Omron Sysmac Studio project Major Project Group 6-week12_011125 (Sysmac Studio 1.56.0.64011, StandardProject)

# Controller new_Controller_0: NX1P2-9024DT1 version 1.64
Task PrimaryTask (priority 4, period or condition 2000): Program0

VAR_GLOBAL
    Start : BOOL;
    PB1 : BOOL;  (* at BuiltInIO://cpu/#0/Input_Bit_08 *)
    PB2 : BOOL;  (* at BuiltInIO://cpu/#0/Input_Bit_09 *)
    PB3 : BOOL;  (* at BuiltInIO://cpu/#0/Input_Bit_10 *)
    PB4 : BOOL;  (* at BuiltInIO://cpu/#0/Input_Bit_11 *)
    LAMP1 : BOOL;  (* Pump On or Off; at BuiltInIO://cpu/#0/Output_Bit_06 *)
    LAMP2 : BOOL;  (* Valve Maintainance; at BuiltInIO://cpu/#0/Output_Bit_07 *)
    LAMP3 : BOOL;  (* at BuiltInIO://cpu/#0/Output_Bit_08 *)
    LAMP4 : BOOL;  (* UV Filter ON or Off; at BuiltInIO://cpu/#0/Output_Bit_09 *)
    Stop : BOOL;
    CYL1 : BOOL;
    CYL2 : BOOL;
    CYL3 : BOOL;
    CYL4 : BOOL;
    CYL1_Retracted : BOOL;  (* at BuiltInIO://cpu/#0/Input_Bit_00 *)
    CYL1_Extended : BOOL;  (* at BuiltInIO://cpu/#0/Input_Bit_01 *)
    CYL2_Retracted : BOOL;  (* at BuiltInIO://cpu/#0/Input_Bit_02 *)
    CYL3_Retracted : BOOL;  (* at BuiltInIO://cpu/#0/Input_Bit_04 *)
    CYL4_Retracted : BOOL;  (* at BuiltInIO://cpu/#0/Input_Bit_06 *)
    CYL2_Extended : BOOL;  (* at BuiltInIO://cpu/#0/Input_Bit_03 *)
    CYL3_Extended : BOOL;  (* at BuiltInIO://cpu/#0/Input_Bit_05 *)
    CYL4_Extended : BOOL;  (* at BuiltInIO://cpu/#0/Input_Bit_07 *)
    CYL1_Retract : BOOL;  (* Valve 1 Open; at BuiltInIO://cpu/#0/Output_Bit_01 *)
    CYL1_Extend : BOOL;  (* Valve 1 Close; at BuiltInIO://cpu/#0/Output_Bit_00 *)
    CYL2_Extend : BOOL;  (* Valve 2 Close; at BuiltInIO://cpu/#0/Output_Bit_02 *)
    CYL3_Extend : BOOL;  (* Valve 3 Close; at BuiltInIO://cpu/#0/Output_Bit_03 *)
    CYL3_Retract : BOOL;  (* Valve 3 Open; at BuiltInIO://cpu/#0/Output_Bit_04 *)
    CYL4_Extend : BOOL;  (* Valve 4 Close; at BuiltInIO://cpu/#0/Output_Bit_05 *)
    CycleRun : BOOL;
    CycleReady : BOOL;
    CylExtendFinish : BOOL;
    CylExtend : BOOL;
    cylRetract : BOOL;
    CylRetractFinish : BOOL;
    CYL2_Retract : BOOL;  (* Valve 2 open *)
    CYL4_Retract : BOOL;  (* Valve 4 Open *)
    Manual_CYL1EXTSignal : BOOL;
    Manual_CYL2EXTSignal : BOOL;
    Manual_CYL3EXTSignal : BOOL;
    Manual_CYL4EXTSignal : BOOL;
    Manual_CYL4RETSignal : BOOL;
    HMI_PB1 : BOOL;
    HMI_PB2 : BOOL;
    HMI_PB3 : BOOL;
    HMI_PB4 : BOOL;
    seqNumber : INT;
    Manual_1 : BOOL;
    Auto_1 : BOOL;
    Manual_2 : BOOL;
    Auto_2 : BOOL;
    Manual_3 : BOOL;
    Auto_3 : BOOL;
    Manual_4 : BOOL;
    Auto_4 : BOOL;
    On_all : BOOL;
    Of_all : BOOL;
    Off_all : BOOL;
    CylSpeed : INT;
    T1_On : TIME;  (* (2000ms) *)
    Pump1_Trip : BOOL;
    StopBotton : BOOL;  (* Manual Pump Off *)
    count1 : INT;
    Valve2Trip : BOOL;
    memory : BOOL;  (* PB1 SW1 Status *)
    memory2 : BOOL;  (* CYL1 SW2 Status *)
    StopBotton1 : BOOL;
    T2_Off : TIME;
    T3_Off : TIME;
    TC1_On : TIME;
    TC2_On : TIME;
    Pump_Status : BOOL;  (* ON/OFF SW P1 *)
    Input2 : BOOL;
    LSW_Low : BOOL;  (* WL Low T1 *)
    LSW_High : BOOL;  (* WL High T1 *)
    Pressure_High : BOOL;
    Pressure_InRange : BOOL;
    Temp_High : BOOL;
    LSW2_High : BOOL;
    LSW2_InRange : BOOL;
    Input10 : BOOL;
    Input11 : BOOL;
    ResetV4 : BOOL;
    ResetV2 : BOOL;
    ResetV3 : BOOL;
    ResetV1 : BOOL;
    System_Test : BOOL;
    Input1 : BOOL;
    V1_Timer : TIME;
    V2_Timer : TIME;
    P1_Off : TIME;
    UV_ON : TIME;
    V3_close : TIME;
    V3_Open : TIME;
    V1_cycle : INT;
    V2_cycle : INT;
    V3_cycle : INT;
    V4_cycle : INT;
    tempOnce : BOOL;
    Cooling : TIME;
    tempTwice : BOOL;
    Count_Cooling : INT;
    Input3 : TIME;
    Input4 : TIME;
    Input5 : TIME;
    Input6 : TIME;
    Input7 : TIME;
    Input8 : TIME;
    Input_10 : TIME;
    Input_11 : TIME;
    Input12 : TIME;
    Input13 : TIME;
    Input14 : TIME;
    Input15 : TIME;
    Input_16 : TIME;
    Input_1 : TIME;
    Input_2 : TIME;
    Cooling2 : TIME;
    V_M : TIME;
    current_countsys : INT;
    System_Checkdone : BOOL;
    V_M4 : TIME;
    check : BOOL;
    Test_Completed : BOOL;
    test_ctu : INT;
    reset_test : BOOL;
    reset_temp : BOOL;
    TestLamp1 : BOOL;
    Test_timer_L4 : TIME;
END_VAR

PROGRAM Program0
VAR
    Ready : BOOL;
    timer_100ms : TON;
    PBDelay : TIME := T#500ms;
    timer1_100ms : TON;
    timer2_100ms : TON;
    timer3_100ms : TON;
    timer4_100ms : TON;
    timer11_100ms : TON;
    timer22_100ms : TON;
    timer33_100ms : TON;
    timer44_100ms : TON;
    Cycler : CTD;
    ResetCtrUp : BOOL;
    CtrUp : CTU;
    CycleTimer : TON;
    CycleTimerOff : TON;
    c_on : BOOL;
    c_off : BOOL;
    c_on_stat : BOOL;
    CycleTimer2 : TON;
    cyl1_off : BOOL;
    cyl2_off : BOOL;
    cyl3_off : BOOL;
    cyl4_off : BOOL;
    auto : BOOL;
    toff4_500ms : TOF;
    toff1_500ms : TOF;
    toff2_500ms : TOF;
    toff3_500ms : TOF;
    PBDownDelay : TIME := T#200ms;
    CylTimer : TIME;
    On_delay_pump : TON;
    Pump_On_Off : CTU;
    T : TOF;
    On_delay_CYL1 : TON;
    On_delay_CYL2 : TON;
    off_delay_valve1 : TOF;
    Off_delay_valve2 : TOF;
    On_delay_pump_SB : TON;
    ON_delay_UV : TON;
    Off_delay_Valve3 : TOF;
    On_delay_valve4 : TON;
    CTU_V1 : CTU;
    CTU_V2 : CTU;
    CTU_V3 : CTU;
    CTU_V4 : CTU;
    On_delay_Cooling : TON;
    CTU_Cooling : CTU;
    I1 : TON;
    I2 : TON;
    I3 : TON;
    I4 : TON;
    I5 : TON;
    I6 : TON;
    I7 : TON;
    I8 : TON;
    I10 : TON;
    I11 : TON;
    I12 : TON;
    I13 : TON;
    I14 : TON;
    I15 : TON;
    I16 : TON;
    OFF_cooling : TOF;
    Valve_Maintance : TP;
    Valve_Maintance1 : TP;
    Count_test : CTD;
    Valve_Maintance2 : TP;
    Valve_Maintance3 : TP;
    Valve_Maintance4 : TP;
    Valve_Maintance5 : TP;
    Valve_Maintance6 : TP;
    Valve_Maintance7 : TP;
    Test_1 : CTU;
    test_comp_time : TON;
    Test_delay_L4 : TON;
    lamp4_on : TIME;
    Systest_on_delay : TON;
END_VAR
VAR_EXTERNAL
    Start : BOOL;
    PB1 : BOOL;
    LAMP1 : BOOL;
    PB2 : BOOL;
    LAMP2 : BOOL;
    PB3 : BOOL;
    LAMP3 : BOOL;
    PB4 : BOOL;
    LAMP4 : BOOL;
    Stop : BOOL;
    CYL1 : BOOL;
    CYL2 : BOOL;
    CYL3 : BOOL;
    CYL4 : BOOL;
    CYL1_Extend : BOOL;
    CYL1_Retract : BOOL;
    CYL2_Extend : BOOL;
    CYL3_Retract : BOOL;
    CYL3_Extend : BOOL;
    CYL4_Extend : BOOL;
    CYL1_Extended : BOOL;
    CycleRun : BOOL;
    CycleReady : BOOL;
    CYL2_Extended : BOOL;
    CYL3_Extended : BOOL;
    CYL4_Extended : BOOL;
    CylExtendFinish : BOOL;
    CylExtend : BOOL;
    CylRetract : BOOL;
    CYL2_Retracted : BOOL;
    CYL3_Retracted : BOOL;
    CYL4_Retracted : BOOL;
    CylRetractFinish : BOOL;
    CYL1_Retracted : BOOL;
    CYL2_Retract : BOOL;
    CYL4_Retract : BOOL;
    Manual_CYL1EXTSignal : BOOL;
    Manual_CYL2EXTSignal : BOOL;
    Manual_CYL3EXTSignal : BOOL;
    Manual_CYL4EXTSignal : BOOL;
    Manual_CYL4RETSignal : BOOL;
    HMI_PB1 : BOOL;
    HMI_PB2 : BOOL;
    HMI_PB3 : BOOL;
    HMI_PB4 : BOOL;
    seqNumber : INT;
    Manual_1 : BOOL;
    Auto_1 : BOOL;
    Manual_2 : BOOL;
    Auto_2 : BOOL;
    Manual_3 : BOOL;
    Auto_3 : BOOL;
    Manual_4 : BOOL;
    Auto_4 : BOOL;
    On_all : BOOL;
    Of_all : BOOL;
    Off_all : BOOL;
    CylSpeed : INT;
    T1_On : TIME;
    Pump1_Trip : BOOL;
    StopBotton : BOOL;
    count1 : INT;
    Valve2Trip : BOOL;
    memory : BOOL;
    memory2 : BOOL;
    StopBotton1 : BOOL;
    T2_Off : TIME;
    T3_Off : TIME;
    TC1_On : TIME;
    TC2_On : TIME;
    LSW_Low : BOOL;
    LSW_High : BOOL;
    Pressure_High : BOOL;
    Pressure_InRange : BOOL;
    Temp_High : BOOL;
    LSW2_High : BOOL;
    LSW2_InRange : BOOL;
    Input10 : BOOL;
    Input11 : BOOL;
    ResetV4 : BOOL;
    ResetV2 : BOOL;
    ResetV3 : BOOL;
    ResetV1 : BOOL;
    System_Test : BOOL;
    Pump_Status : BOOL;
    Input1 : BOOL;
    V1_Timer : TIME;
    V2_Timer : TIME;
    P1_Off : TIME;
    UV_ON : TIME;
    V3_close : TIME;
    V3_Open : TIME;
    V1_cycle : INT;
    V2_cycle : INT;
    V3_cycle : INT;
    V4_cycle : INT;
    tempOnce : BOOL;
    Cooling : TIME;
    tempTwice : BOOL;
    Count_Cooling : INT;
    Input2 : BOOL;
    Input3 : TIME;
    Input4 : TIME;
    Input5 : TIME;
    Input6 : TIME;
    Input7 : TIME;
    Input8 : TIME;
    Input_10 : TIME;
    Input_11 : TIME;
    Input12 : TIME;
    Input13 : TIME;
    Input14 : TIME;
    Input15 : TIME;
    Input_16 : TIME;
    Input_1 : TIME;
    Input_2 : TIME;
    Cooling2 : TIME;
    V_M : TIME;
    current_countsys : INT;
    System_Checkdone : BOOL;
    V_M4 : TIME;
    check : BOOL;
    Test_Completed : BOOL;
    test_ctu : INT;
    reset_test : BOOL;
    reset_temp : BOOL;
    TestLamp1 : BOOL;
    Test_timer_L4 : TIME;
END_VAR
VAR
    _e1 : R_TRIG;
    _e2 : R_TRIG;
    _e3 : R_TRIG;
    _e4 : R_TRIG;
    _e5 : R_TRIG;
    _e6 : R_TRIG;
END_VAR

(* Section Main_Program: ladder, written here as Structured Text *)

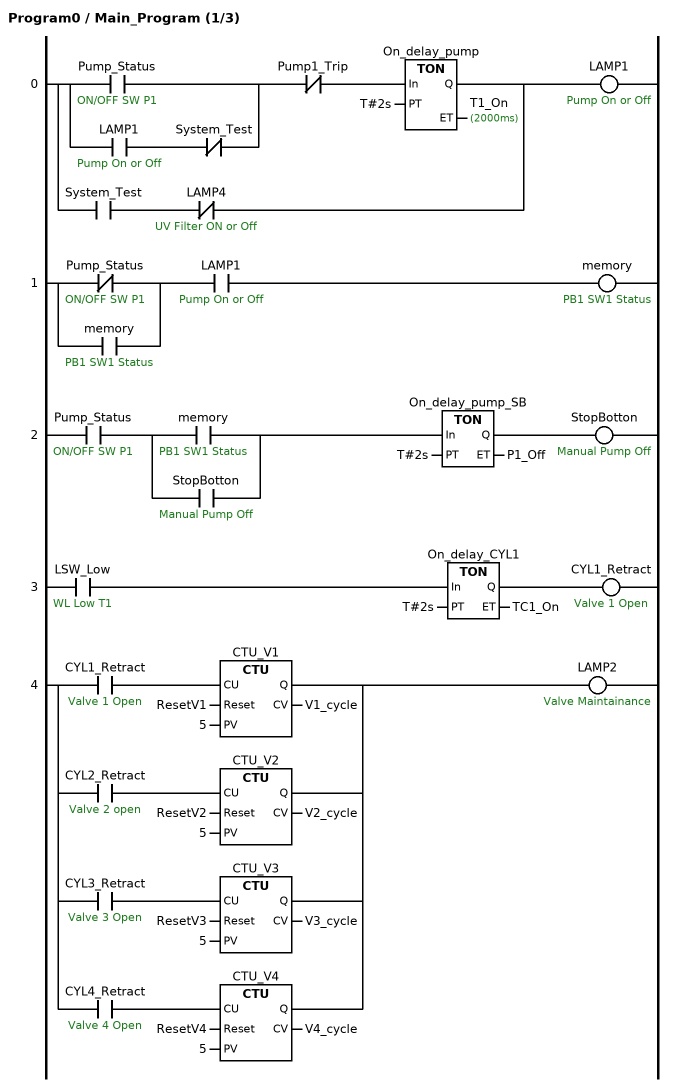
(* Rung 0 *)
On_delay_pump(In := (Pump_Status OR (LAMP1 AND NOT System_Test)) AND NOT Pump1_Trip, PT := T#2s, ET => T1_On);
LAMP1 := On_delay_pump.Q OR (System_Test AND NOT LAMP4);
(* Rung 1 *)
memory := (NOT Pump_Status OR memory) AND LAMP1;
(* Rung 2 *)
On_delay_pump_SB(In := Pump_Status AND (memory OR StopBotton), PT := T#2s, ET => P1_Off);
StopBotton := On_delay_pump_SB.Q;
(* Rung 3 *)
On_delay_CYL1(In := LSW_Low, PT := T#2s, ET => TC1_On);
CYL1_Retract := On_delay_CYL1.Q;
(* Rung 4 *)
_e1(CLK := CYL1_Retract);
CTU_V1(CU := _e1.Q, Reset := ResetV1, PV := 5, CV => V1_cycle);
_e2(CLK := CYL2_Retract);
CTU_V2(CU := _e2.Q, Reset := ResetV2, PV := 5, CV => V2_cycle);
_e3(CLK := CYL3_Retract);
CTU_V3(CU := _e3.Q, Reset := ResetV3, PV := 5, CV => V3_cycle);
_e4(CLK := CYL4_Retract);
CTU_V4(CU := _e4.Q, Reset := ResetV4, PV := 5, CV => V4_cycle);
LAMP2 := CTU_V1.Q OR CTU_V2.Q OR CTU_V3.Q OR CTU_V4.Q;

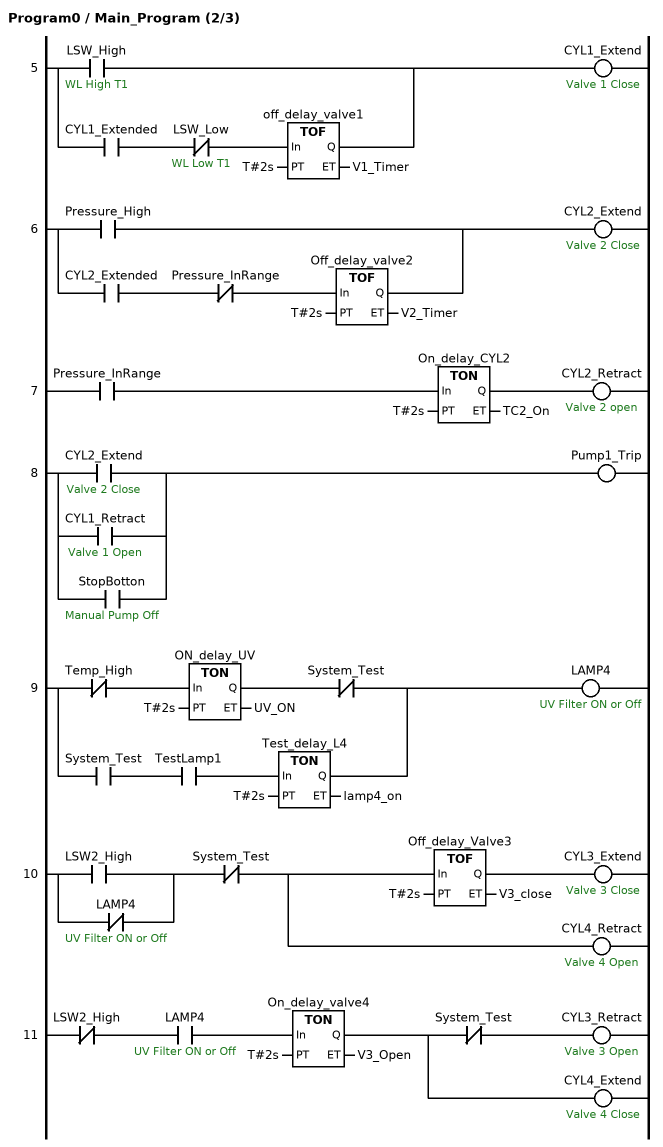
(* Rung 5 *)
off_delay_valve1(In := CYL1_Extended AND NOT LSW_Low, PT := T#2s, ET => V1_Timer);
CYL1_Extend := LSW_High OR off_delay_valve1.Q;
(* Rung 6 *)
Off_delay_valve2(In := CYL2_Extended AND NOT Pressure_InRange, PT := T#2s, ET => V2_Timer);
CYL2_Extend := Pressure_High OR Off_delay_valve2.Q;
(* Rung 7 *)
On_delay_CYL2(In := Pressure_InRange, PT := T#2s, ET => TC2_On);
CYL2_Retract := On_delay_CYL2.Q;
(* Rung 8 *)
Pump1_Trip := CYL2_Extend OR CYL1_Retract OR StopBotton;
(* Rung 9 *)
ON_delay_UV(In := NOT Temp_High, PT := T#2s, ET => UV_ON);
Test_delay_L4(In := System_Test AND TestLamp1, PT := T#2s, ET => lamp4_on);
LAMP4 := (ON_delay_UV.Q AND NOT System_Test) OR Test_delay_L4.Q;
(* Rung 10 *)
Off_delay_Valve3(In := (LSW2_High OR NOT LAMP4) AND NOT System_Test, PT := T#2s, ET => V3_close);
CYL3_Extend := Off_delay_Valve3.Q;
CYL4_Retract := (LSW2_High OR NOT LAMP4) AND NOT System_Test;
(* Rung 11 *)
On_delay_valve4(In := NOT LSW2_High AND LAMP4, PT := T#2s, ET => V3_Open);
CYL3_Retract := On_delay_valve4.Q AND NOT System_Test;
CYL4_Extend := On_delay_valve4.Q;

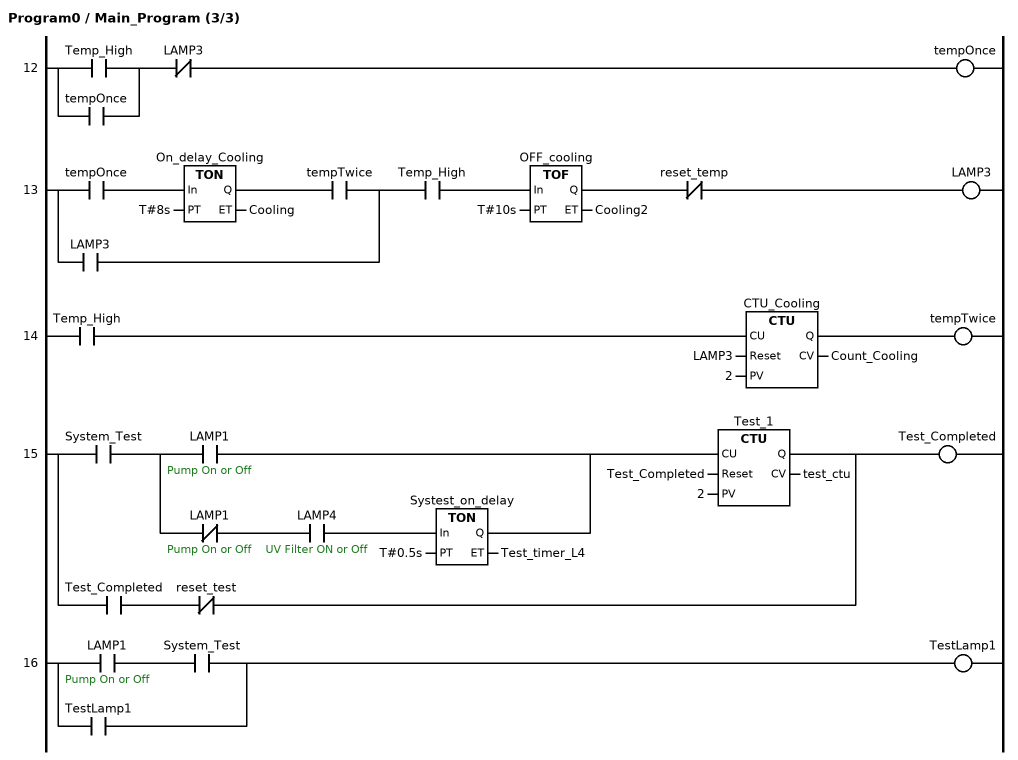
(* Rung 12 *)
tempOnce := (Temp_High OR tempOnce) AND NOT LAMP3;
(* Rung 13 *)
On_delay_Cooling(In := tempOnce, PT := T#8s, ET => Cooling);
OFF_cooling(In := ((On_delay_Cooling.Q AND tempTwice) OR LAMP3) AND Temp_High, PT := T#10s, ET => Cooling2);
LAMP3 := OFF_cooling.Q AND NOT reset_temp;
(* Rung 14 *)
_e5(CLK := Temp_High);
CTU_Cooling(CU := _e5.Q, Reset := LAMP3, PV := 2, CV => Count_Cooling);
tempTwice := CTU_Cooling.Q;
(* Rung 15 *)
Systest_on_delay(In := System_Test AND NOT LAMP1 AND LAMP4, PT := T#0.5s, ET => Test_timer_L4);
_e6(CLK := (System_Test AND LAMP1) OR Systest_on_delay.Q);
Test_1(CU := _e6.Q, Reset := Test_Completed, PV := 2, CV => test_ctu);
Test_Completed := Test_1.Q OR (Test_Completed AND NOT reset_test);
(* Rung 16 *)
TestLamp1 := (LAMP1 AND System_Test) OR TestLamp1;

(* Section Input_Combination: ladder, written here as Structured Text *)

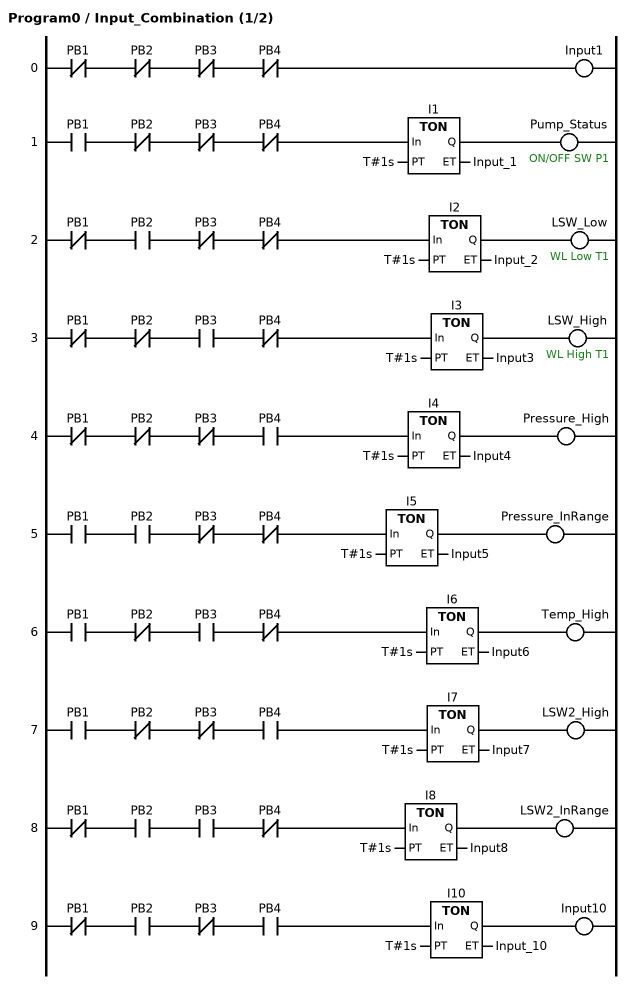
(* Rung 0 *)
Input1 := NOT PB1 AND NOT PB2 AND NOT PB3 AND NOT PB4;
(* Rung 1 *)
I1(In := PB1 AND NOT PB2 AND NOT PB3 AND NOT PB4, PT := T#1s, ET => Input_1);
Pump_Status := I1.Q;
(* Rung 2 *)
I2(In := NOT PB1 AND PB2 AND NOT PB3 AND NOT PB4, PT := T#1s, ET => Input_2);
LSW_Low := I2.Q;
(* Rung 3 *)
I3(In := NOT PB1 AND NOT PB2 AND PB3 AND NOT PB4, PT := T#1s, ET => Input3);
LSW_High := I3.Q;
(* Rung 4 *)
I4(In := NOT PB1 AND NOT PB2 AND NOT PB3 AND PB4, PT := T#1s, ET => Input4);
Pressure_High := I4.Q;
(* Rung 5 *)
I5(In := PB1 AND PB2 AND NOT PB3 AND NOT PB4, PT := T#1s, ET => Input5);
Pressure_InRange := I5.Q;
(* Rung 6 *)
I6(In := PB1 AND NOT PB2 AND PB3 AND NOT PB4, PT := T#1s, ET => Input6);
Temp_High := I6.Q;
(* Rung 7 *)
I7(In := PB1 AND NOT PB2 AND NOT PB3 AND PB4, PT := T#1s, ET => Input7);
LSW2_High := I7.Q;
(* Rung 8 *)
I8(In := NOT PB1 AND PB2 AND PB3 AND NOT PB4, PT := T#1s, ET => Input8);
LSW2_InRange := I8.Q;
(* Rung 9 *)
I10(In := NOT PB1 AND PB2 AND NOT PB3 AND PB4, PT := T#1s, ET => Input_10);
Input10 := I10.Q;

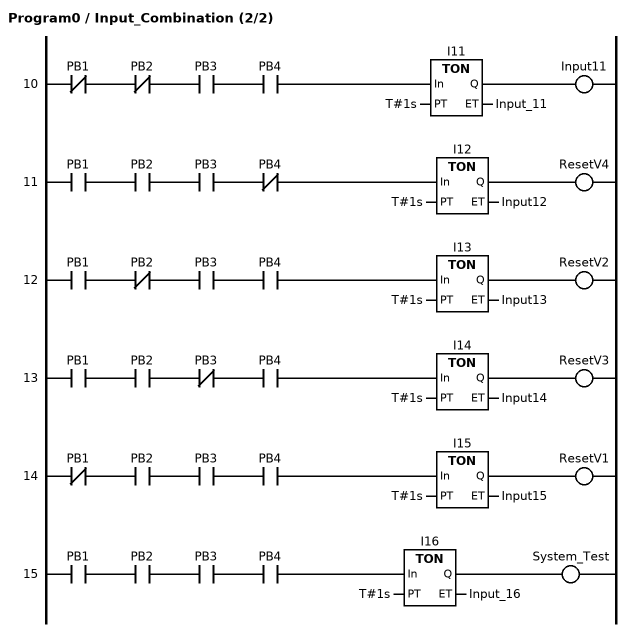
(* Rung 10 *)
I11(In := NOT PB1 AND NOT PB2 AND PB3 AND PB4, PT := T#1s, ET => Input_11);
Input11 := I11.Q;
(* Rung 11 *)
I12(In := PB1 AND PB2 AND PB3 AND NOT PB4, PT := T#1s, ET => Input12);
ResetV4 := I12.Q;
(* Rung 12 *)
I13(In := PB1 AND NOT PB2 AND PB3 AND PB4, PT := T#1s, ET => Input13);
ResetV2 := I13.Q;
(* Rung 13 *)
I14(In := PB1 AND PB2 AND NOT PB3 AND PB4, PT := T#1s, ET => Input14);
ResetV3 := I14.Q;
(* Rung 14 *)
I15(In := NOT PB1 AND PB2 AND PB3 AND PB4, PT := T#1s, ET => Input15);
ResetV1 := I15.Q;
(* Rung 15 *)
I16(In := PB1 AND PB2 AND PB3 AND PB4, PT := T#1s, ET => Input_16);
System_Test := I16.Q;
END_PROGRAM

# Device HMI_NA5_0 (NA): not converted